(* PLC project 02_task_and_scopes.project, CODESYS CODESYS V3.5 SP22 Patch 2 *)
(* stored: creationDateTime 2026-07-23T05:49:24.5434818, modificationDateTime 2026-07-23T05:48:41.9165944 *)

PROGRAM PLC_PRG
  VAR
    xRunning : BOOL := FALSE;  (* Running Coil *)
  END_VAR

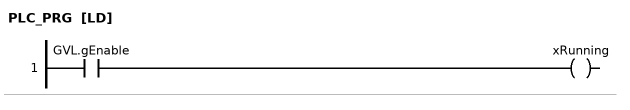
(* LD diagram, written out as Structured Text *)
(* Random comment for this program *)

xRunning := GVL.gEnable;
END_PROGRAM

CONFIGURATION Application
  RESOURCE Application ON PLC
    {attribute 'qualified_only'}
    VAR_GLOBAL  (* GVL *)
      gEnable : BOOL;
      gRunCount : DINT;
    END_VAR
    TASK MainTask(INTERVAL := T#20ms, PRIORITY := 1);
    PROGRAM PLC_PRG WITH MainTask : PLC_PRG;
  END_RESOURCE
END_CONFIGURATION
